FUNCTION RadToDeg : REAL

VAR_INPUT
	fAngle : REAL;
END_VAR

VAR
	fRadToDegConstant : REAL := 57.295;
END_VAR

VAR_OUTPUT
	fAngleDeg : REAL;
END_VAR


fAngleDeg := fAngle * fRadToDegConstant;

END_FUNCTION

(* stored: Version 1.1.0.1, ProductVersion 3.1.4024.12
   POU RadToDeg: Id {7f79deb0-186c-47c5-b496-96e4697c7c77}, SpecialFunc None *)
